// TIA Portal V17 export
// export: Created 2025-03-05T08:00:12.2598366Z, ExportSetting WithDefaults, DisplayName Totally Integrated Automation Portal, DisplayVersion V17 Update 8, DisplayName TIA Portal Openness, DisplayVersion V17 Update 8, DisplayName TIA Portal Version Control Interface, DisplayVersion V17, DisplayName SINAMICS Startdrive Advanced, DisplayVersion V17 SP2, DisplayName SINAMICS Startdrive G110M, G120, G120C, G120D, G120P, G115D, DisplayVersion V17 SP2, DisplayName SINAMICS Startdrive G130, G150, S120, S150, SINAMICS MV, S210, DisplayVersion V17 SP2, DisplayName STEP 7 Professional, DisplayVersion V17 Update 8, DisplayName SINUMERIK ONE STEP 7 Toolbox, DisplayVersion V17 Update 12, DisplayName SINUMERIK 840D sl STEP 7 Toolbox, DisplayVersion V17 Update 12, DisplayName STEP 7 Safety, DisplayVersion V17 Update 6, DisplayName WinCC Advanced, DisplayVersion V17 Update 8
FUNCTION "FC2109_STATION_3_LIGHT_U01" : Void   // FC2109, LAD
{ S7_Optimized_Access := 'FALSE' }
AUTHOR : ETXETAR
VERSION : 1.0
// stored: AutoNumber false, IsIECCheckEnabled false, SetENOAutomatically false, UDAEnableTagReadback false
   VAR_TEMP   // added for the SCL form of the ladder/FBD networks
      _w1 : Bool;
   END_VAR
BEGIN

REGION Network 1: INPUTS
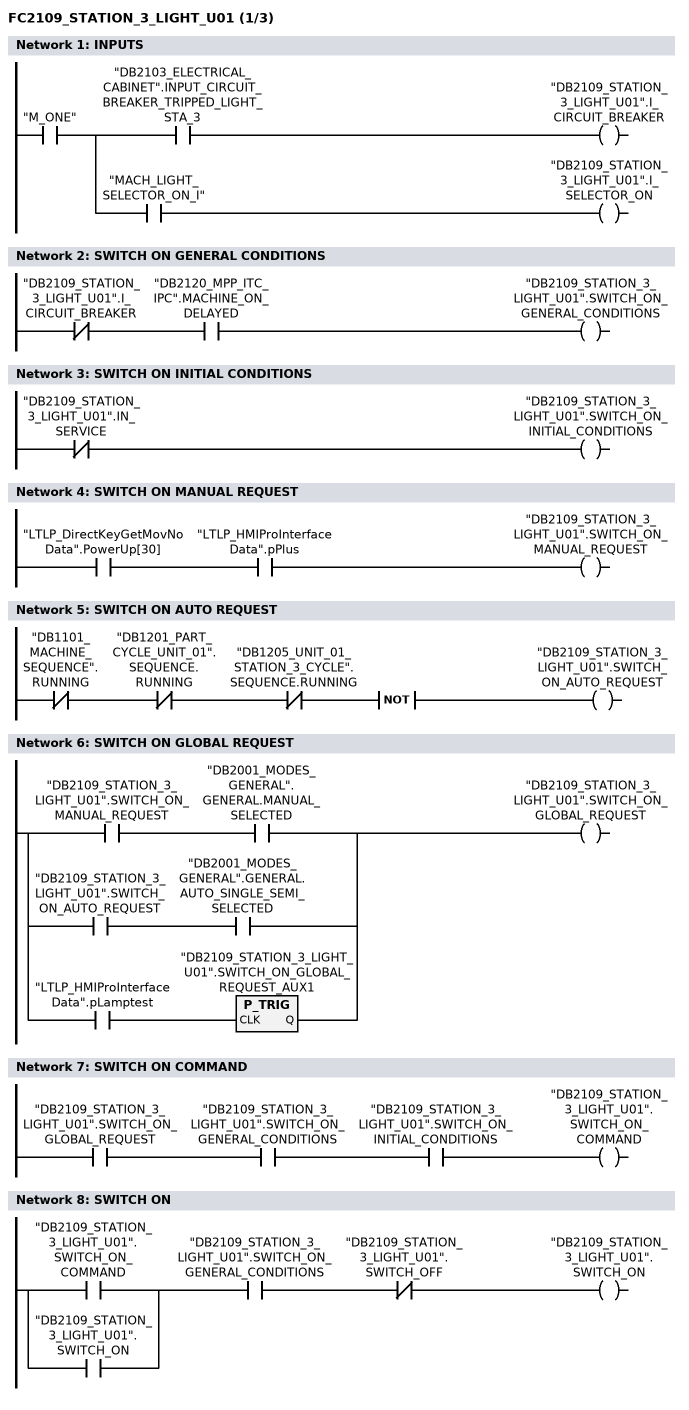
   RUNG wire#powerrail
      Contact( "M_ONE" )
      wire#w1
      Contact( "DB2103_ELECTRICAL_CABINET".INPUT_CIRCUIT_BREAKER_TRIPPED_LIGHT_STA_3 )
      Coil( "DB2109_STATION_3_LIGHT_U01".I_CIRCUIT_BREAKER )
   END_RUNG
   RUNG wire#w1
      Contact( "MACH_LIGHT_SELECTOR_ON_I" )
      Coil( "DB2109_STATION_3_LIGHT_U01".I_SELECTOR_ON )
   END_RUNG
   // the same network as SCL:
   "DB2109_STATION_3_LIGHT_U01".I_CIRCUIT_BREAKER := "M_ONE" AND "DB2103_ELECTRICAL_CABINET".INPUT_CIRCUIT_BREAKER_TRIPPED_LIGHT_STA_3;
   "DB2109_STATION_3_LIGHT_U01".I_SELECTOR_ON := "M_ONE" AND "MACH_LIGHT_SELECTOR_ON_I";
END_REGION

REGION Network 2: SWITCH ON GENERAL CONDITIONS
   RUNG wire#powerrail
      I_Contact( "DB2109_STATION_3_LIGHT_U01".I_CIRCUIT_BREAKER )
      Contact( "DB2120_MPP_ITC_IPC".MACHINE_ON_DELAYED )
      Coil( "DB2109_STATION_3_LIGHT_U01".SWITCH_ON_GENERAL_CONDITIONS )
   END_RUNG
   // the same network as SCL:
   "DB2109_STATION_3_LIGHT_U01".SWITCH_ON_GENERAL_CONDITIONS := NOT "DB2109_STATION_3_LIGHT_U01".I_CIRCUIT_BREAKER AND "DB2120_MPP_ITC_IPC".MACHINE_ON_DELAYED;
END_REGION

REGION Network 3: SWITCH ON INITIAL CONDITIONS
   RUNG wire#powerrail
      I_Contact( "DB2109_STATION_3_LIGHT_U01".IN_SERVICE )
      Coil( "DB2109_STATION_3_LIGHT_U01".SWITCH_ON_INITIAL_CONDITIONS )
   END_RUNG
   // the same network as SCL:
   "DB2109_STATION_3_LIGHT_U01".SWITCH_ON_INITIAL_CONDITIONS := NOT "DB2109_STATION_3_LIGHT_U01".IN_SERVICE;
END_REGION

REGION Network 4: SWITCH ON MANUAL REQUEST
   RUNG wire#powerrail
      Contact( "LTLP_DirectKeyGetMovNoData".PowerUp[30] )
      Contact( "LTLP_HMIProInterfaceData".pPlus )
      Coil( "DB2109_STATION_3_LIGHT_U01".SWITCH_ON_MANUAL_REQUEST )
   END_RUNG
   // the same network as SCL:
   "DB2109_STATION_3_LIGHT_U01".SWITCH_ON_MANUAL_REQUEST := "LTLP_DirectKeyGetMovNoData".PowerUp[30] AND "LTLP_HMIProInterfaceData".pPlus;
END_REGION

REGION Network 5: SWITCH ON AUTO REQUEST
   RUNG wire#powerrail
      I_Contact( "DB1101_MACHINE_SEQUENCE".RUNNING )
      I_Contact( "DB1201_PART_CYCLE_UNIT_01".SEQUENCE.RUNNING )
      I_Contact( "DB1205_UNIT_01_STATION_3_CYCLE".SEQUENCE.RUNNING )
      Not()
      Coil( "DB2109_STATION_3_LIGHT_U01".SWITCH_ON_AUTO_REQUEST )
   END_RUNG
   // the same network as SCL:
   "DB2109_STATION_3_LIGHT_U01".SWITCH_ON_AUTO_REQUEST := NOT (NOT "DB1101_MACHINE_SEQUENCE".RUNNING AND NOT "DB1201_PART_CYCLE_UNIT_01".SEQUENCE.RUNNING AND NOT "DB1205_UNIT_01_STATION_3_CYCLE".SEQUENCE.RUNNING);
END_REGION

REGION Network 6: SWITCH ON GLOBAL REQUEST
   RUNG wire#powerrail
      Contact( "DB2109_STATION_3_LIGHT_U01".SWITCH_ON_MANUAL_REQUEST )
      Contact( "DB2001_MODES_GENERAL".GENERAL.MANUAL_SELECTED )
      wire#w1
      Coil( "DB2109_STATION_3_LIGHT_U01".SWITCH_ON_GLOBAL_REQUEST )
   END_RUNG
   RUNG wire#powerrail
      Contact( "DB2109_STATION_3_LIGHT_U01".SWITCH_ON_AUTO_REQUEST )
      Contact( "DB2001_MODES_GENERAL".GENERAL.AUTO_SINGLE_SEMI_SELECTED )
   END_RUNG wire#w1
   RUNG wire#powerrail
      Contact( "LTLP_HMIProInterfaceData".pLamptest )
      P_Trig( "DB2109_STATION_3_LIGHT_U01".SWITCH_ON_GLOBAL_REQUEST_AUX1 )
   END_RUNG wire#w1
   // the same network as SCL:
   #_w1 := "LTLP_HMIProInterfaceData".pLamptest AND NOT "DB2109_STATION_3_LIGHT_U01".SWITCH_ON_GLOBAL_REQUEST_AUX1;   // rising edge
   "DB2109_STATION_3_LIGHT_U01".SWITCH_ON_GLOBAL_REQUEST_AUX1 := "LTLP_HMIProInterfaceData".pLamptest;
   "DB2109_STATION_3_LIGHT_U01".SWITCH_ON_GLOBAL_REQUEST := ("DB2109_STATION_3_LIGHT_U01".SWITCH_ON_MANUAL_REQUEST AND "DB2001_MODES_GENERAL".GENERAL.MANUAL_SELECTED) OR ("DB2109_STATION_3_LIGHT_U01".SWITCH_ON_AUTO_REQUEST AND "DB2001_MODES_GENERAL".GENERAL.AUTO_SINGLE_SEMI_SELECTED) OR #_w1;
END_REGION

REGION Network 7: SWITCH ON COMMAND
   RUNG wire#powerrail
      Contact( "DB2109_STATION_3_LIGHT_U01".SWITCH_ON_GLOBAL_REQUEST )
      Contact( "DB2109_STATION_3_LIGHT_U01".SWITCH_ON_GENERAL_CONDITIONS )
      Contact( "DB2109_STATION_3_LIGHT_U01".SWITCH_ON_INITIAL_CONDITIONS )
      Coil( "DB2109_STATION_3_LIGHT_U01".SWITCH_ON_COMMAND )
   END_RUNG
   // the same network as SCL:
   "DB2109_STATION_3_LIGHT_U01".SWITCH_ON_COMMAND := "DB2109_STATION_3_LIGHT_U01".SWITCH_ON_GLOBAL_REQUEST AND "DB2109_STATION_3_LIGHT_U01".SWITCH_ON_GENERAL_CONDITIONS AND "DB2109_STATION_3_LIGHT_U01".SWITCH_ON_INITIAL_CONDITIONS;
END_REGION

REGION Network 8: SWITCH ON
   RUNG wire#powerrail
      Contact( "DB2109_STATION_3_LIGHT_U01".SWITCH_ON_COMMAND )
      wire#w1
      Contact( "DB2109_STATION_3_LIGHT_U01".SWITCH_ON_GENERAL_CONDITIONS )
      I_Contact( "DB2109_STATION_3_LIGHT_U01".SWITCH_OFF )
      Coil( "DB2109_STATION_3_LIGHT_U01".SWITCH_ON )
   END_RUNG
   RUNG wire#powerrail
      Contact( "DB2109_STATION_3_LIGHT_U01".SWITCH_ON )
   END_RUNG wire#w1
   // the same network as SCL:
   "DB2109_STATION_3_LIGHT_U01".SWITCH_ON := ("DB2109_STATION_3_LIGHT_U01".SWITCH_ON_COMMAND OR "DB2109_STATION_3_LIGHT_U01".SWITCH_ON) AND "DB2109_STATION_3_LIGHT_U01".SWITCH_ON_GENERAL_CONDITIONS AND NOT "DB2109_STATION_3_LIGHT_U01".SWITCH_OFF;
END_REGION

REGION Network 9: IN SERVICE
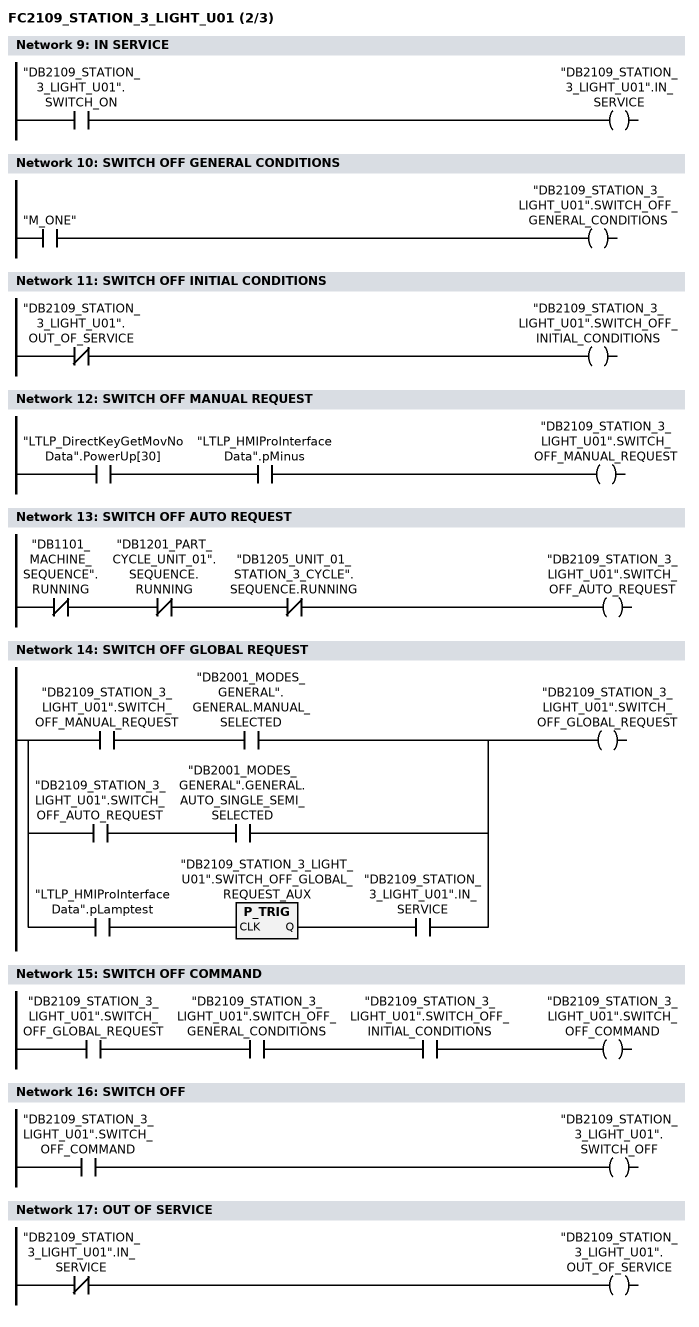
   RUNG wire#powerrail
      Contact( "DB2109_STATION_3_LIGHT_U01".SWITCH_ON )
      Coil( "DB2109_STATION_3_LIGHT_U01".IN_SERVICE )
   END_RUNG
   // the same network as SCL:
   "DB2109_STATION_3_LIGHT_U01".IN_SERVICE := "DB2109_STATION_3_LIGHT_U01".SWITCH_ON;
END_REGION

REGION Network 10: SWITCH OFF GENERAL CONDITIONS
   RUNG wire#powerrail
      Contact( "M_ONE" )
      Coil( "DB2109_STATION_3_LIGHT_U01".SWITCH_OFF_GENERAL_CONDITIONS )
   END_RUNG
   // the same network as SCL:
   "DB2109_STATION_3_LIGHT_U01".SWITCH_OFF_GENERAL_CONDITIONS := "M_ONE";
END_REGION

REGION Network 11: SWITCH OFF INITIAL CONDITIONS
   RUNG wire#powerrail
      I_Contact( "DB2109_STATION_3_LIGHT_U01".OUT_OF_SERVICE )
      Coil( "DB2109_STATION_3_LIGHT_U01".SWITCH_OFF_INITIAL_CONDITIONS )
   END_RUNG
   // the same network as SCL:
   "DB2109_STATION_3_LIGHT_U01".SWITCH_OFF_INITIAL_CONDITIONS := NOT "DB2109_STATION_3_LIGHT_U01".OUT_OF_SERVICE;
END_REGION

REGION Network 12: SWITCH OFF MANUAL REQUEST
   RUNG wire#powerrail
      Contact( "LTLP_DirectKeyGetMovNoData".PowerUp[30] )
      Contact( "LTLP_HMIProInterfaceData".pMinus )
      Coil( "DB2109_STATION_3_LIGHT_U01".SWITCH_OFF_MANUAL_REQUEST )
   END_RUNG
   // the same network as SCL:
   "DB2109_STATION_3_LIGHT_U01".SWITCH_OFF_MANUAL_REQUEST := "LTLP_DirectKeyGetMovNoData".PowerUp[30] AND "LTLP_HMIProInterfaceData".pMinus;
END_REGION

REGION Network 13: SWITCH OFF AUTO REQUEST
   RUNG wire#powerrail
      I_Contact( "DB1101_MACHINE_SEQUENCE".RUNNING )
      I_Contact( "DB1201_PART_CYCLE_UNIT_01".SEQUENCE.RUNNING )
      I_Contact( "DB1205_UNIT_01_STATION_3_CYCLE".SEQUENCE.RUNNING )
      Coil( "DB2109_STATION_3_LIGHT_U01".SWITCH_OFF_AUTO_REQUEST )
   END_RUNG
   // the same network as SCL:
   "DB2109_STATION_3_LIGHT_U01".SWITCH_OFF_AUTO_REQUEST := NOT "DB1101_MACHINE_SEQUENCE".RUNNING AND NOT "DB1201_PART_CYCLE_UNIT_01".SEQUENCE.RUNNING AND NOT "DB1205_UNIT_01_STATION_3_CYCLE".SEQUENCE.RUNNING;
END_REGION

REGION Network 14: SWITCH OFF GLOBAL REQUEST
   RUNG wire#powerrail
      Contact( "DB2109_STATION_3_LIGHT_U01".SWITCH_OFF_MANUAL_REQUEST )
      Contact( "DB2001_MODES_GENERAL".GENERAL.MANUAL_SELECTED )
      wire#w1
      Coil( "DB2109_STATION_3_LIGHT_U01".SWITCH_OFF_GLOBAL_REQUEST )
   END_RUNG
   RUNG wire#powerrail
      Contact( "DB2109_STATION_3_LIGHT_U01".SWITCH_OFF_AUTO_REQUEST )
      Contact( "DB2001_MODES_GENERAL".GENERAL.AUTO_SINGLE_SEMI_SELECTED )
   END_RUNG wire#w1
   RUNG wire#powerrail
      Contact( "LTLP_HMIProInterfaceData".pLamptest )
      P_Trig( "DB2109_STATION_3_LIGHT_U01".SWITCH_OFF_GLOBAL_REQUEST_AUX )
      Contact( "DB2109_STATION_3_LIGHT_U01".IN_SERVICE )
   END_RUNG wire#w1
   // the same network as SCL:
   #_w1 := "LTLP_HMIProInterfaceData".pLamptest AND NOT "DB2109_STATION_3_LIGHT_U01".SWITCH_OFF_GLOBAL_REQUEST_AUX;   // rising edge
   "DB2109_STATION_3_LIGHT_U01".SWITCH_OFF_GLOBAL_REQUEST_AUX := "LTLP_HMIProInterfaceData".pLamptest;
   "DB2109_STATION_3_LIGHT_U01".SWITCH_OFF_GLOBAL_REQUEST := ("DB2109_STATION_3_LIGHT_U01".SWITCH_OFF_MANUAL_REQUEST AND "DB2001_MODES_GENERAL".GENERAL.MANUAL_SELECTED) OR ("DB2109_STATION_3_LIGHT_U01".SWITCH_OFF_AUTO_REQUEST AND "DB2001_MODES_GENERAL".GENERAL.AUTO_SINGLE_SEMI_SELECTED) OR (#_w1 AND "DB2109_STATION_3_LIGHT_U01".IN_SERVICE);
END_REGION

REGION Network 15: SWITCH OFF COMMAND
   RUNG wire#powerrail
      Contact( "DB2109_STATION_3_LIGHT_U01".SWITCH_OFF_GLOBAL_REQUEST )
      Contact( "DB2109_STATION_3_LIGHT_U01".SWITCH_OFF_GENERAL_CONDITIONS )
      Contact( "DB2109_STATION_3_LIGHT_U01".SWITCH_OFF_INITIAL_CONDITIONS )
      Coil( "DB2109_STATION_3_LIGHT_U01".SWITCH_OFF_COMMAND )
   END_RUNG
   // the same network as SCL:
   "DB2109_STATION_3_LIGHT_U01".SWITCH_OFF_COMMAND := "DB2109_STATION_3_LIGHT_U01".SWITCH_OFF_GLOBAL_REQUEST AND "DB2109_STATION_3_LIGHT_U01".SWITCH_OFF_GENERAL_CONDITIONS AND "DB2109_STATION_3_LIGHT_U01".SWITCH_OFF_INITIAL_CONDITIONS;
END_REGION

REGION Network 16: SWITCH OFF
   RUNG wire#powerrail
      Contact( "DB2109_STATION_3_LIGHT_U01".SWITCH_OFF_COMMAND )
      Coil( "DB2109_STATION_3_LIGHT_U01".SWITCH_OFF )
   END_RUNG
   // the same network as SCL:
   "DB2109_STATION_3_LIGHT_U01".SWITCH_OFF := "DB2109_STATION_3_LIGHT_U01".SWITCH_OFF_COMMAND;
END_REGION

REGION Network 17: OUT OF SERVICE
   RUNG wire#powerrail
      I_Contact( "DB2109_STATION_3_LIGHT_U01".IN_SERVICE )
      Coil( "DB2109_STATION_3_LIGHT_U01".OUT_OF_SERVICE )
   END_RUNG
   // the same network as SCL:
   "DB2109_STATION_3_LIGHT_U01".OUT_OF_SERVICE := NOT "DB2109_STATION_3_LIGHT_U01".IN_SERVICE;
END_REGION

REGION Network 18: HMI STATUS
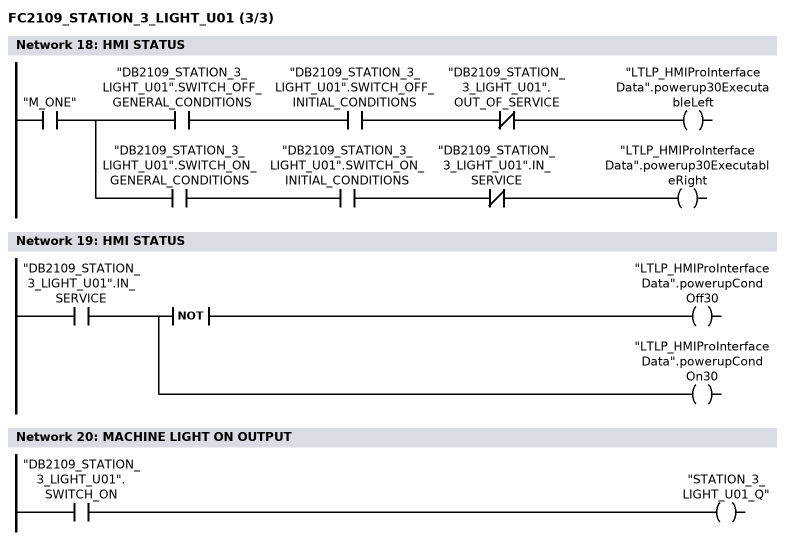
   RUNG wire#powerrail
      Contact( "M_ONE" )
      wire#w1
      Contact( "DB2109_STATION_3_LIGHT_U01".SWITCH_OFF_GENERAL_CONDITIONS )
      Contact( "DB2109_STATION_3_LIGHT_U01".SWITCH_OFF_INITIAL_CONDITIONS )
      I_Contact( "DB2109_STATION_3_LIGHT_U01".OUT_OF_SERVICE )
      Coil( "LTLP_HMIProInterfaceData".powerup30ExecutableLeft )
   END_RUNG
   RUNG wire#w1
      Contact( "DB2109_STATION_3_LIGHT_U01".SWITCH_ON_GENERAL_CONDITIONS )
      Contact( "DB2109_STATION_3_LIGHT_U01".SWITCH_ON_INITIAL_CONDITIONS )
      I_Contact( "DB2109_STATION_3_LIGHT_U01".IN_SERVICE )
      Coil( "LTLP_HMIProInterfaceData".powerup30ExecutableRight )
   END_RUNG
   // the same network as SCL:
   "LTLP_HMIProInterfaceData".powerup30ExecutableLeft := "M_ONE" AND "DB2109_STATION_3_LIGHT_U01".SWITCH_OFF_GENERAL_CONDITIONS AND "DB2109_STATION_3_LIGHT_U01".SWITCH_OFF_INITIAL_CONDITIONS AND NOT "DB2109_STATION_3_LIGHT_U01".OUT_OF_SERVICE;
   "LTLP_HMIProInterfaceData".powerup30ExecutableRight := "M_ONE" AND "DB2109_STATION_3_LIGHT_U01".SWITCH_ON_GENERAL_CONDITIONS AND "DB2109_STATION_3_LIGHT_U01".SWITCH_ON_INITIAL_CONDITIONS AND NOT "DB2109_STATION_3_LIGHT_U01".IN_SERVICE;
END_REGION

REGION Network 19: HMI STATUS
   RUNG wire#powerrail
      Contact( "DB2109_STATION_3_LIGHT_U01".IN_SERVICE )
      wire#w1
      Not()
      Coil( "LTLP_HMIProInterfaceData".powerupCondOff30 )
   END_RUNG
   RUNG wire#w1
      Coil( "LTLP_HMIProInterfaceData".powerupCondOn30 )
   END_RUNG
   // the same network as SCL:
   "LTLP_HMIProInterfaceData".powerupCondOff30 := NOT "DB2109_STATION_3_LIGHT_U01".IN_SERVICE;
   "LTLP_HMIProInterfaceData".powerupCondOn30 := "DB2109_STATION_3_LIGHT_U01".IN_SERVICE;
END_REGION

REGION Network 20: MACHINE LIGHT ON OUTPUT
   RUNG wire#powerrail
      Contact( "DB2109_STATION_3_LIGHT_U01".SWITCH_ON )
      Coil( "STATION_3_LIGHT_U01_Q" )
   END_RUNG
   // the same network as SCL:
   "STATION_3_LIGHT_U01_Q" := "DB2109_STATION_3_LIGHT_U01".SWITCH_ON;
END_REGION
END_FUNCTION
